FUNCTION_BLOCK PUBLIC FB_Axis IMPLEMENTS ITF_Axis
VAR
	testString : STRING;
END_VAR

METHOD Disable : BOOL
VAR_INPUT
END_VAR
ADSLOGSTR( msgCtrlMask := ADSLOG_MSGTYPE_ERROR OR ADSLOG_MSGTYPE_MSGBOX,
			msgFmtStr :='Axis Disabling',
 			strArg := '');
END_METHOD

METHOD Enable : BOOL
VAR_INPUT
	EnablePositive : BOOL;
	EnableNegative : BOOL;
	Override : LREAL;
END_VAR
testString := '';
testString := CONCAT(testString, '[');
testString := CONCAT(testString, BOOL_TO_STRING(EnablePositive));
testString := CONCAT(testString, ']');
testString := CONCAT(testString, '[');
testString := CONCAT(testString, BOOL_TO_STRING(EnableNegative));
testString := CONCAT(testString, ']');
testString := CONCAT(testString, '[');
testString := CONCAT(testString, LREAL_TO_STRING(Override));
testString := CONCAT(testString, ']');

ADSLOGSTR( msgCtrlMask := ADSLOG_MSGTYPE_ERROR OR ADSLOG_MSGTYPE_MSGBOX,
			msgFmtStr :='Axis Enabling: %s',
 			strArg := testString);
END_METHOD

METHOD MoveToPosition : BOOL
VAR_INPUT
	Position : LREAL;
	Velocity : LREAL;
END_VAR
testString := '';
testString := CONCAT(testString, '[');
testString := CONCAT(testString, LREAL_TO_STRING(Position));
testString := CONCAT(testString, ']');
testString := CONCAT(testString, '[');
testString := CONCAT(testString, LREAL_TO_STRING(Velocity));
testString := CONCAT(testString, ']');

ADSLOGSTR( msgCtrlMask := ADSLOG_MSGTYPE_ERROR OR ADSLOG_MSGTYPE_MSGBOX,
			msgFmtStr :='Axis Moving: %s',
 			strArg := testString);
END_METHOD

END_FUNCTION_BLOCK

(* stored: Version 1.1.0.1, ProductVersion 3.1.4024.12
   POU FB_Axis: Id {4af9d760-2be5-422f-b1a0-874998de53c5}, SpecialFunc None
   Method Disable: Id {61f52bb7-111d-4919-beb3-f9b352c00d02}
   Method Enable: Id {69d6a0ec-a06c-4b17-93fb-ef1ac4c62c7a}
   Method MoveToPosition: Id {70cff655-1362-4500-8eab-04fe4ebf0588} *)
